Staubli VAL3: encodeAck.pgx

public program encodeAck()
begin
  switch rosGenericMsg.header.nMsgType
    case 11
      call encTrajPtAck()
    break
    case 14
      call encTrajPtFAck()
    break
    default
    break
  endSwitch
end
